{attribute 'qualified_only'}
VAR_GLOBAL
	Start: BOOL;
	Stop: BOOL;
	Reset: BOOL;
	Run: BOOL;
	Alarm: BOOL;
	Error: BOOL;	
END_VAR

(* stored: Version 1.1.0.1, ProductVersion 3.1.4024.12
   GVL gHMI: Id {fc4c07f8-6b9d-4642-a312-b22b865d6b70} *)
